FUNCTION_BLOCK FB_Robot
VAR_INPUT
END_VAR
VAR_OUTPUT
END_VAR
VAR
	{attribute 'TcInitSymbol'}
	oidInstance : OTCID;
	ipRobot : IRobot;
	hrInit : HRESULT;
END_VAR

METHOD FB_exit : BOOL
VAR_INPUT
	bInCopyCode : BOOL; // if TRUE, the exit method is called for exiting an instance that is copied afterwards (online change).
END_VAR
IF NOT bInCopyCode THEN
	FW_SafeRelease(ADR(ipRobot));
END_IF
END_METHOD

METHOD FB_init : BOOL
VAR_INPUT
	bInitRetains : BOOL; // if TRUE, the retain variables are initialized (warm start / cold start)
	bInCopyCode : BOOL;  // if TRUE, the instance afterwards gets moved into the copy code (online change)
END_VAR
IF NOT bInCopyCode THEN
	IF ipRobot = 0 THEN
		hrInit := FW_objMgr_GetObjectInstance(oid := oidInstance, iid:= TC_GLOBAL_IID_LIST.IID_IRobot,pipUnk := ADR(ipRobot)); 
	END_IF
END_IF
END_METHOD

{attribute 'c++_compatible'}
{attribute 'minimal_input_size' := '4'}
{attribute 'pack_mode' := '4'}
{warning 'add method implementation'}
METHOD InitRobot : UDINT
VAR_INPUT
	pInitPar	: POINTER TO st_InitParameter;
END_VAR
IF (ipRobot <> 0) THEN
	InitRobot := ipRobot.InitRobot(pInitPar);
END_IF
END_METHOD


{attribute 'c++_compatible'}
{attribute 'minimal_input_size' := '4'}
{attribute 'pack_mode' := '4'}


METHOD RunRobot : UDINT
VAR_INPUT
	pMC_Inputs	: POINTER TO st_AxisGroupRead;
	pMC_Outputs	: POINTER TO st_AxisGroupSet;
	pCtlComd	: POINTER TO Recvbuff;
	pRobotStatus	: POINTER TO Sendbuff;
END_VAR
IF (ipRobot <> 0) THEN
	RunRobot := ipRobot.RunRobot(pMC_Inputs, pMC_Outputs, pCtlComd, pRobotStatus);
END_IF
END_METHOD

{attribute 'c++_compatible'}
{attribute 'minimal_input_size' := '4'}
{attribute 'pack_mode' := '4'}
{warning 'add method implementation'}
METHOD StopRobot : HRESULT
IF (ipRobot <> 0) THEN
	StopRobot := ipRobot.StopRobot();
END_IF
END_METHOD

END_FUNCTION_BLOCK

(* stored: Version 1.1.0.1, ProductVersion 3.1.4022.12
   POU FB_Robot: Id {bb53ae37-266d-444e-acc5-1c032fe98f91}, SpecialFunc None
   Method FB_exit: Id {8ae06666-ce55-4525-94dc-d8d6be7e4422}
   Method FB_init: Id {6d818fef-0880-4cfe-9732-3d632cfc8a37}
   Method InitRobot: Id {e1a75cb4-1f0b-4169-8d34-9e93f166f4f3}
   Method RunRobot: Id {54fbf472-68a6-4ad3-ab8e-f0741a546ddd}
   Method StopRobot: Id {1bd503dc-9449-46d6-87aa-d98db2c4979f} *)
